VAR_GLOBAL
    ads_watch_dog : FB_ADS_WATCHDOG;
    ads_watch_dog_qrix : FB_ADS_WATCHDOG;

    FB_MR3K2_FIM_ILK : FB_EXT_ILK;
    {attribute 'pytmc' := '
        pv: PLC:KFE:RIX:FIM:MR3K2:ILK
    '}
    ST_MR3K2_FIM_ILK : ST_EXT_ILK := (rPRO_SP := 2e-7);
    FB_MR4K2_FIM_ILK : FB_EXT_ILK;
    {attribute 'pytmc' := '
        pv: PLC:KFE:RIX:FIM:MR4K2:ILK
    '}
    ST_MR4K2_FIM_ILK : ST_EXT_ILK := (rPRO_SP := 2e-7);
END_VAR

(* stored: Version 1.1.0.1, ProductVersion 3.1.4022.18
   GVL GVL_RIX_INTF: Id {0a70a95d-d899-4d85-b505-d428da9aa702} *)
